FUNCTION_BLOCK FB_StateCtrlCycleTest_1 EXTENDS FB_MasterArmCtrlBase
VAR_INPUT
END_VAR
VAR_OUTPUT
END_VAR
VAR
	//arm id
	m_armId:INT;			
	
	//test step
	m_testStep:INT:=-1;
	
	//motion parameters
	m_maxjntVel,m_maxjntAcc,m_maxjntJerk:Vec7d;
	
	//time
	m_time:LREAL;
		
	//test point
	m_pointNum:INT;
	
	//motion start
	m_startMotion:BOOL;
	m_startMotionLast:BOOL;
	
	//home position
	m_homeDHPos,m_startDHJntPos,m_endDHJntPos:Vec7d;
	
	//joint position gap
	m_jntDist:Vec7d:=[30.0*g_deg2Rad,20.0*g_deg2Rad,20.0*g_deg2Rad,30.0*g_deg2Rad,30.0*g_deg2Rad,20.0*g_deg2Rad,30.0*g_deg2Rad];
			
	//startJntPos,endJntPos :Vec8d;
	m_initJntPos,m_startJntPos,m_endJntPos :Vec7d;
	
	//motion distance
	m_motDist:Vec7d;
	
	//Trajectory planner
	m_Planner: FB_TrajMoveJ;
	
	//basic function
	m_basicFun:FB_BasicFun;
	
	//unit function
	m_unitFun:FB_UnitTransform;
	
	//target joint position
	m_targetJntPos:ARRAY[1..10] OF Vec7d;
	
	//point sum
	m_pointSum:INT;
	
	//target cycle number
	m_motionCycleNum:INT;
	m_targetCycleNum:INT;
	
	//cycle time
	m_curCycleTime:LREAL;
	
	//current DH joint position
	m_curDHJntPos:Vec7d;
END_VAR

// override this function in each exact controller
METHOD PROTECTED calcCmdJntPos : BOOL

VAR_IN_OUT CONSTANT
	i_slaveIdx :INT;
	i_shoulderPose :ST_Frame;
	i_masterArm :FB_MasterArm;
	i_slaveStatus :ST_SlaveStatus;
END_VAR

//joint enable
m_jntEnableFlag :=g_cycleTest.m_jntEnable[i_masterArm.armIdx];

//init parameters flag
IF (g_cycleTest.m_enterESDTest[m_armId]=TRUE) THEN
	m_startMotion:=TRUE;
ELSE
	m_startMotion:=g_cycleTest.m_startMotion[m_armId];	
END_IF

//monitoring signal rising edge
IF (m_startMotionLast=FALSE) AND (m_startMotion=TRUE)THEN
	m_testStep:=0;
END_IF
m_startMotionLast:=m_startMotion;

//frequency test and step test
testMotion(i_masterArm);

//update the information
updateInfo(i_masterArm);



//******************data for monitor which can be deleted**********************//
GVL_Monitor.g_stateMachine[m_armId]:=MasterArmControl.m_masterRobot.m_masterArmState[m_armId];
GVL_Monitor.g_jntPos[m_armId]:=i_masterArm.curJntPos;
GVL_Monitor.g_step[m_armId]:=m_testStep;
GVL_Monitor.g_time[m_armId]:=m_time;
GVL_Monitor.g_targetPos[m_armId]:=m_cmdJntPos;
GVL_Monitor.g_pointNum[m_armId]:=m_pointNum;
END_METHOD

// override this function in each exact controller
// NOTICE: set joint control mode here, and do some initialization if needed
METHOD PUBLIC init : BOOL
VAR_IN_OUT CONSTANT
	i_masterArm	:FB_MasterArm;
END_VAR
VAR_IN_OUT 
	r_masterArmCtrlCmd :ST_ArmCtrlCmds;
END_VAR

VAR
	i:INT;
END_VAR

SUPER^.Init(i_masterArm,r_masterArmCtrlCmd);
copyCmds(r_masterArmCtrlCmd);


//variable initialization
m_armId:=i_masterArm.armIdx;
m_startMotionLast:=FALSE;

//joint enable
g_cycleTest.m_jntEnable[m_armId]:=g_onesVec7i;


//velocity---acceleration---jerk
vecMultiNum(GVL_ArmJointParameters.g_maxJntVel,0.1,m_maxjntVel);
vecMultiNum(m_maxjntVel,3,m_maxjntAcc);
vecMultiNum(m_maxjntAcc,3,m_maxjntJerk);


//joint home position---joint motion start position and end position
FOR i:=1 TO g_mJntNum BY 1 DO
	m_homeDHPos[i]:=gvl_const.g_jntDHInitPos[m_armId,i];
	m_jntDist[i]:=10.0*g_deg2Rad;
	m_startDHJntPos[i]:=m_homeDHPos[i]-m_jntDist[i];
	m_endDHJntPos[i]:=m_homeDHPos[i]+m_jntDist[i];	
END_FOR


//variable test point number
IF (g_cycleTest.m_enterESDTest[m_armId]=FALSE) THEN
	m_pointSum:=g_cycleTest.m_pointSum[m_armId];
	m_targetCycleNum:=g_cycleTest.m_targetCycleNum[m_armId];
	FOR i:=1 TO 10 BY 1 DO
		m_targetJntPos[i]:=m_unitFun.masterArmUnit2System(i_dataTest:= g_cycleTest.m_targetJntPos[m_armId,i]);
	END_FOR	
ELSE
	m_pointSum:=3;
	m_targetCycleNum:=30000;
	m_targetJntPos[1]:=m_startDHJntPos; 	m_targetJntPos[2]:=m_homeDHPos;	m_targetJntPos[3]:=m_endDHJntPos;
END_IF
END_METHOD

METHOD testMotion : BOOL
VAR_INPUT
	i_masterArm :FB_MasterArm;
END_VAR

VAR
	i:INT;
	//DH joint position
	startDHPos,endDHPos,targetDHPos :Vec7d;
	r_masterArmCtrlCmd :ST_ArmCtrlCmds;
END_VAR

CASE m_testStep OF
	0: //init
		IF (g_cycleTest.m_enterESDTest[m_armId]=FALSE) THEN
			m_pointSum:=g_cycleTest.m_pointSum[m_armId];
			m_targetCycleNum:=g_cycleTest.m_targetCycleNum[m_armId];
			FOR i:=1 TO 10 BY 1 DO
				m_targetJntPos[i]:=m_unitFun.masterArmUnit2System(i_dataTest:= g_cycleTest.m_targetJntPos[m_armId,i]);
			END_FOR
		ELSE
			g_cycleTest.m_tgtCycleTime[m_armId]:=10;
		END_IF
		
		m_maxjntVel:=m_unitFun.masterArmUnit2System(i_dataTest:=g_cycleTest.m_targetJntVel[m_armId]);
		FOR i:=1 TO 7 BY 1 DO			
			IF ABS(m_maxjntVel[i])<g_smallNum THEN
				m_maxjntVel[i]:=1;
			END_IF
			m_maxjntVel[i]:=LIMIT(-GVL_ArmJointParameters.g_maxJntVel[i],m_maxjntVel[i],GVL_ArmJointParameters.g_maxJntVel[i]);
		END_FOR
		vecMultiNum(m_maxjntVel,3,m_maxjntAcc);
		vecMultiNum(m_maxjntAcc,3,m_maxjntJerk);
		
		m_pointNum:=1;	
		m_motionCycleNum:=0;	
		m_curCycleTime:=0;
		m_testStep:=10;
		
		
	10: //Trajectory parameter initialization
		m_basicFun.activeJnt2DH(i_activeJntPos:= i_masterArm.curJntPos, o_DHJntPos=> startDHPos);		
		endDHPos:=m_targetJntPos[m_pointNum];	
		
		//limit the joint position
		FOR i:=1 TO 7 BY 1 DO
			startDHPos[i]:=LIMIT(gvl_const.g_minJntDHPos[m_armId,i],startDHPos[i],gvl_const.g_maxJntDHPos[m_armId,i]);
			endDHPos[i]:=LIMIT(gvl_const.g_minJntDHPos[m_armId,i],endDHPos[i],gvl_const.g_maxJntDHPos[m_armId,i]);
		END_FOR
		
		//motion distance judgement
		vecSub(endDHPos,startDHPos,m_motDist);
		IF (norm(m_motDist)<g_smallNum) THEN
			m_testStep:=25;
			RETURN;
		END_IF
		
		m_Planner.init(i_startJntPos:= startDHPos, 	i_targetJntPos:= endDHPos, 	i_maxJntVel:= m_maxjntVel, 	i_maxJntAcc:= m_maxjntAcc, 	i_maxJntJerk:= m_maxjntJerk);
		IF (m_Planner.isGene=FALSE) THEN
			m_testStep:=30;
		ELSE
			m_time:=0; m_testStep:=20;
		END_IF
		
		
	20: //start motion
		IF (g_cycleTest.m_pause[m_armId]=TRUE) THEN
			//g_cycleTest.m_pause[m_armId]:=FALSE;
			RETURN;
		END_IF
		
		IF (g_cycleTest.m_finish[m_armId]=TRUE) THEN
			g_cycleTest.m_finish[m_armId]:=FALSE;
			m_testStep:=30;
			RETURN;
		END_IF
		
		//motion duration
		m_time:=m_time+g_armCtrlCycleTime;
		m_Planner.evaluate(t:= m_time, jntPos=> targetDHPos, jntVel=> m_cmdJntVel, jntAcc=> m_cmdJntAcc);
		m_basicFun.DH2activeJnt(i_DHJntPos:= targetDHPos, o_activeJntPos=> m_cmdJntPos);		
		IF (m_time>m_Planner.duration) THEN
			m_testStep:=25;			
		END_IF		
		
		//end the motion
		IF (m_startMotion=FALSE) THEN
			m_testStep:=30;
		END_IF
		
		
	25: //Record the motion cycle
		m_pointNum:=m_pointNum+1;
		IF (m_pointNum>m_pointSum) THEN
			m_pointNum:=1;
			m_motionCycleNum:=m_motionCycleNum+1;
			//IF (m_motionCycleNum>m_targetCycleNum) THEN
			IF (g_cycleTest.m_curCycleTime[m_armId]>g_cycleTest.m_tgtCycleTime[m_armId]) THEN
				m_testStep:=30;
			ELSE
				m_testStep:=10;
			END_IF
		ELSE
			m_testStep:=10;
		END_IF	
		
		
	30: //end the motion
		m_testStep:=-1;		
END_CASE
m_curCycleTime:=m_curCycleTime+g_armCtrlCycleTime;


//feedback the information to ui
g_cycleTest.m_curPointNum[m_armId]:=m_pointNum;
g_cycleTest.m_curCycleNum[m_armId]:=m_motionCycleNum;
g_cycleTest.m_curCycleTime[m_armId]:=m_curCycleTime/3600;
END_METHOD

METHOD updateInfo : BOOL
VAR_INPUT
	i_masterArm :FB_MasterArm;
END_VAR

VAR
	i:INT;
	targetJntPos:Vec7d;
END_VAR

//update the joint position
FOR i:=1 TO g_mJntNum BY 1 DO
	g_cycleTest.m_motorEncoder[m_armId][i]:=i_masterArm.m_joints[i].m_motorInputs.m_motorEncoder;
	g_cycleTest.m_jntEncoder[m_armId][i]:=i_masterArm.m_joints[i].m_motorInputs.m_linkEncoder;
END_FOR

//g_cycleTest.m_armActJntPos[m_armId]:=i_masterArm.curJntPos;
g_cycleTest.m_armActJntPos[m_armId]:=m_unitFun.masterArmUnit2User(i_dataSystem:= i_masterArm.curJntPos);
m_basicFun.activeJnt2DH(i_activeJntPos:= i_masterArm.curJntPos, o_DHJntPos=> m_curDHJntPos);
g_cycleTest.m_armDHJntPos[m_armId]:=m_unitFun.masterArmUnit2User(i_dataSystem:= m_curDHJntPos);

//cover the target joint position
IF (g_cycleTest.m_coverCmdPos[m_armId]=TRUE) THEN
	i:=g_cycleTest.m_pntIdForCoverCmd[m_armId];
	IF (i>=1) AND (i<=10) THEN
		g_cycleTest.m_targetJntPos[m_armId,i]:=g_cycleTest.m_armDHJntPos[m_armId];
		m_targetJntPos[i]:=g_cycleTest.m_armDHJntPos[m_armId];
	END_IF
END_IF
END_METHOD

END_FUNCTION_BLOCK

(* stored: Version 1.1.0.1, ProductVersion 3.1.4024.11
   POU FB_StateCtrlCycleTest_1: Id {e378f210-355c-4300-b17a-c04b422ac67a}, SpecialFunc None
   Method calcCmdJntPos: Id {5e3f1fcd-9e7d-4661-b76c-629b047948e0}
   Method init: Id {e8390fa7-0573-41a8-8422-575c47a8c2a8}
   Method testMotion: Id {abc49800-b5f7-40ba-9c65-a5718af0c017}
   Method updateInfo: Id {90e32b55-be07-4352-b89a-e83bf9f90cc7} *)
